TYPE ST_EtherCatSyncUnitTaskInfo :
	STRUCT
		WcState	   : BIT;
		ObjectId   : OTCID;
		State	   : UINT;
		SlaveCount : UINT;
	END_STRUCT
END_TYPE

(* stored: Version 1.1.0.1, ProductVersion 3.1.4026.18
   DUT ST_EtherCatSyncUnitTaskInfo: Id {1ad3ce28-8764-0f5f-29ce-da927a859126} *)
